// TIA Portal V17 export
// export: Created 2024-08-13T13:17:37.5625193Z, ExportSetting WithDefaults, DisplayName Totally Integrated Automation Portal, DisplayVersion V17 Update 5, DisplayName TIA Portal Openness, DisplayVersion V17 Update 5, DisplayName TIA Portal Version Control Interface, DisplayVersion V17, DisplayName SINAMICS Startdrive Advanced, DisplayVersion V17 SP1, DisplayName SINAMICS Startdrive G130, G150, S120, S150, SINAMICS MV, S210, DisplayVersion V17 SP1, DisplayName SINAMICS Startdrive G110M, G120, G120C, G120D, G120P, G115D, DisplayVersion V17 SP1, DisplayName STEP 7 Professional, DisplayVersion V17 Update 5, DisplayName STEP 7 Safety, DisplayVersion V17, DisplayName WinCC Advanced / Unified PC, DisplayVersion V17 Update 5
FUNCTION "GS1_MODBUS" : Void   // FC1, LAD
TITLE = FUNCTION FOR SEND THE MODE (R/W OF REGISTERS), MODBUS MODE, REGISTERS ADDRESS AND LOAD VALUES
{ S7_Optimized_Access := 'TRUE' }
VERSION : 0.1
// stored: AutoNumber true, IsIECCheckEnabled false, SetENOAutomatically false, UDAEnableTagReadback false
   VAR_OUTPUT
      GS1_DONE : Bool;
      GS1_BUSY : Bool;
      GS1_ERROR : Bool;
      GS1_STATUS : Word;
   END_VAR
   VAR_TEMP   // added for the SCL form of the ladder/FBD networks
      _w1 : Bool;
   END_VAR
BEGIN

REGION Network 1: ----------[GENERATE MODBUS ADDRESS & COMMAND DATA INDEX]----------
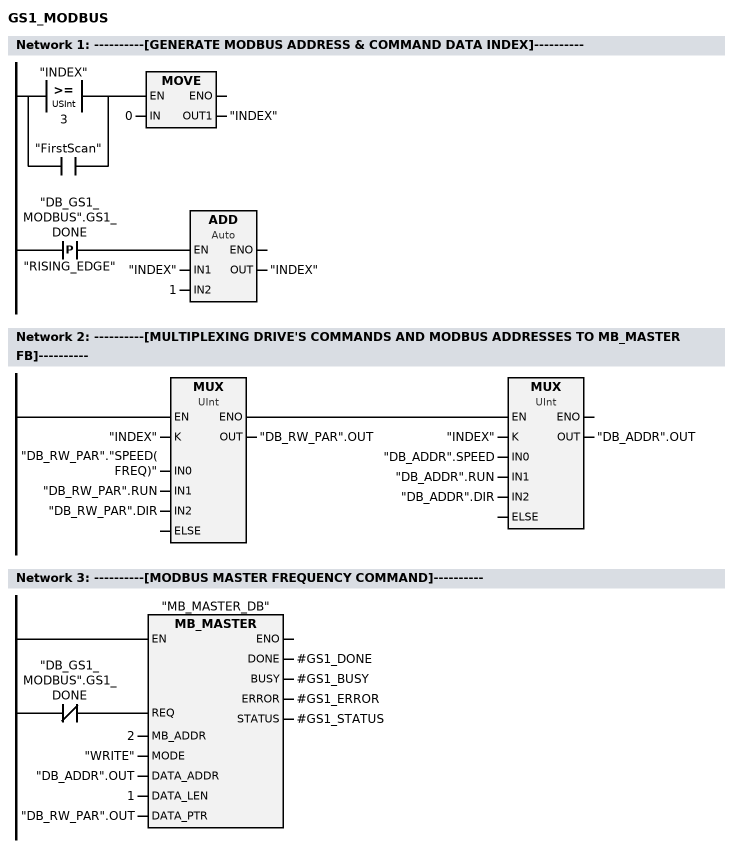
   RUNG wire#powerrail
      { S7_Templates := "SrcType := USInt" } GE_Contact(in1 := "INDEX", in2 := 3)
      wire#w1
      Move(in := 0, out1 => "INDEX")
   END_RUNG
   RUNG wire#powerrail
      Contact( "FirstScan" )
   END_RUNG wire#w1
   RUNG wire#powerrail
      P_Contact(operand := "DB_GS1_MODBUS".GS1_DONE, bit := "RISING_EDGE")
      Add(in1 := "INDEX", in2 := 1, out => "INDEX")
   END_RUNG
   // the same network as SCL:
   IF ("INDEX" >= 3) OR "FirstScan" THEN "INDEX" := 0; END_IF;
   #_w1 := "DB_GS1_MODBUS".GS1_DONE AND NOT "RISING_EDGE";   // rising edge of "DB_GS1_MODBUS".GS1_DONE
   "RISING_EDGE" := "DB_GS1_MODBUS".GS1_DONE;
   IF #_w1 THEN "INDEX" := "INDEX" + 1; END_IF;
END_REGION

REGION Network 2: ----------[MULTIPLEXING DRIVE'S COMMANDS AND MODBUS ADDRESSES TO MB_MASTER FB]----------
   RUNG wire#powerrail
      { S7_Templates := "SrcType := UInt"; S7_GenerateENO := "TRUE" } Mux(k := "INDEX", in0 := "DB_RW_PAR"."SPEED(FREQ)", in1 := "DB_RW_PAR".RUN, in2 := "DB_RW_PAR".DIR, "else" :=, out => "DB_RW_PAR".OUT)
      { S7_Templates := "SrcType := UInt"; S7_GenerateENO := "TRUE" } Mux(k := "INDEX", in0 := "DB_ADDR".SPEED, in1 := "DB_ADDR".RUN, in2 := "DB_ADDR".DIR, "else" :=, out => "DB_ADDR".OUT)
   END_RUNG
   // the same network as SCL:
   // no SCL statement known for Mux: written as a call
   // ENO of a box is taken as its EN; it also drops when the box reports an error
   Mux(k := "INDEX",
       in0 := "DB_RW_PAR"."SPEED(FREQ)",
       in1 := "DB_RW_PAR".RUN,
       in2 := "DB_RW_PAR".DIR,
       out => "DB_RW_PAR".OUT);
   Mux(k := "INDEX", in0 := "DB_ADDR".SPEED, in1 := "DB_ADDR".RUN, in2 := "DB_ADDR".DIR, out => "DB_ADDR".OUT);
END_REGION

REGION Network 3: ----------[MODBUS MASTER FREQUENCY COMMAND]----------
   RUNG wire#powerrail
      "MB_MASTER_DB".MB_MASTER(REQ := wire#w1, MB_ADDR := 2, MODE := "WRITE", DATA_ADDR := "DB_ADDR".OUT, DATA_LEN := 1, DATA_PTR := "DB_RW_PAR".OUT, DONE => #GS1_DONE, BUSY => #GS1_BUSY, ERROR => #GS1_ERROR, STATUS => #GS1_STATUS)
   END_RUNG
   RUNG wire#powerrail
      I_Contact( "DB_GS1_MODBUS".GS1_DONE )
   END_RUNG wire#w1
   // the same network as SCL:
   "MB_MASTER_DB"(REQ := NOT "DB_GS1_MODBUS".GS1_DONE,   // MB_MASTER
                  MB_ADDR := 2,
                  MODE := "WRITE",
                  DATA_ADDR := "DB_ADDR".OUT,
                  DATA_LEN := 1,
                  DATA_PTR := "DB_RW_PAR".OUT,
                  DONE => #GS1_DONE,
                  BUSY => #GS1_BUSY,
                  ERROR => #GS1_ERROR,
                  STATUS => #GS1_STATUS);
END_REGION
END_FUNCTION
